FUNCTION_BLOCK FB_GenericUPS IMPLEMENTS iUPS
VAR_INPUT
END_VAR
VAR_OUTPUT
END_VAR
VAR
END_VAR

{warning 'add method implementation '}
METHOD persist_data : BOOL
END_METHOD

{warning 'add method implementation '}
METHOD shutdown : BOOL
END_METHOD

{warning 'add property implementation'}
PROPERTY UPSState : E_UPSState
GET
END_GET
SET
END_SET
END_PROPERTY

{warning 'add method implementation '}
METHOD watch_status : BOOL
END_METHOD

END_FUNCTION_BLOCK

(* stored: Version 1.1.0.1, ProductVersion 3.1.4024.12
   POU FB_GenericUPS: Id {cde44bd3-bf34-4547-83d5-45e53bbe73f8}, SpecialFunc None
   Method persist_data: Id {45ab1615-aefd-4eef-999b-6783725b4f04}
   Method shutdown: Id {ce1cc227-402c-4d0d-af5a-1144c1ce391e}
   Property UPSState: Id {977c4584-2f65-4f58-b857-efd1b92807d1}
   Get Get: Id {b43077a2-2c3d-43c9-9c09-5b01941b8326}
   Set Set: Id {484f989f-8554-4520-a8da-7a44326dd89f}
   Method watch_status: Id {3d777f1e-d591-44f5-b313-af2e7cf7a433} *)
